FUNCTION_BLOCK FB_PositionStateMove_Test EXTENDS TcUnit.FB_TestSuite
VAR
    Expected: BOOL := True;
    Actual: BOOL;
END_VAR

TEST('FB_PositionStateMove_Test Dummy Test');
AssertEquals(Expected := Expected,
             Actual := Actual,
             Message := 'Error Message');
TEST_FINISHED();

END_FUNCTION_BLOCK

(* stored: Version 1.1.0.1, ProductVersion 3.1.4022.18
   POU FB_PositionStateMove_Test: Id {06e29f1b-dd79-4a48-99b4-9f1a0953646e}, SpecialFunc None *)
